TYPE "typeAngleInputParam"
VERSION : 0.1
   STRUCT
      filterTimeConsts : Array[1.."AXIS_NUM"] of Real;
      scalingParams : Array[1.."AXIS_NUM"] of "typeScaleParam";
   END_STRUCT;

END_TYPE

